TYPE
    ST_TableMoveStatus EXTENDS ST_ServiceStatus_Base :
    STRUCT
    END_STRUCT
END_TYPE

(* stored: Version 1.1.0.1, ProductVersion 3.1.4024.13
   DUT ST_TableMoveStatus: Id {b5b538c5-84b6-4a1b-865f-40e0d54a6314} *)
